{attribute addProperty BoxType "EKM1101-0000-0016"}
{attribute addProperty Id "ControlAT %Q*Control_24A93024162"}
{attribute addProperty CRC "968972988"}
{attribute addProperty SizeInBites "16"}
{attribute addProperty SizeInBytes "2"}
TYPE MMS_Device_Outputs_39C15ABC :
STRUCT
	{attribute addProperty Name "Control"}
	Control AT %Q* : Control_24A93024;
END_STRUCT
END_TYPE

(* stored: Version 1.2.0.0, ProductVersion 3.1.4024.9
   DUT MMS_Device_Outputs_39C15ABC: Id {99a51cef-b6d5-411b-af65-2fe6fc730559} *)
